FUNCTION_BLOCK pi (* 1st ordem system *)
  (* Standard: 61499-2 *)
  (* Version 11-01-12, GASR *)
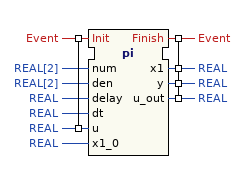
  EVENT_INPUT
    Init WITH u;
  END_EVENT
  EVENT_OUTPUT
    Finish WITH x1, y, u_out;
  END_EVENT
  VAR_INPUT
    num : ARRAY [0..1] OF REAL;
    den : ARRAY [0..1] OF REAL;
    delay : REAL := 0;
    dt : REAL;
    u : REAL;
    x1_0 : REAL; (* condicao inicial *)
  END_VAR
  VAR_OUTPUT
    x1 : REAL;
    y : REAL;
    u_out : REAL;
  END_VAR
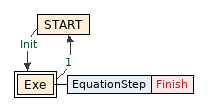
  EC_STATES
    Exe : EquationStep -> Finish;
    START;
  END_STATES
  EC_TRANSITIONS
    Exe TO START := 1;
    START TO Exe := Init;
  END_TRANSITIONS
  ALGORITHM EquationStep IN Lua: (* den[1] = b0, den[2] = b1 *)

						if type(input_buffer) ~= 'table' then
							input_buffer = {}
							for i = 1, math.ceil(delay/dt) +2 do
								input_buffer[#input_buffer +1] = 0
							end
						end
						input_buffer[#input_buffer] = u
						u = input_buffer[1]
						for i = 1, #input_buffer-1 do
							input_buffer[i] = input_buffer[i+1]
						end

						local beta1 = (num[2] - den[2]*num[1])

						local function f1(X1, U)
							return -den[2]*X1 + beta1*U
						end


						R11 = dt*f1(x1_0, u);
						x1aux = x1_0 + 0.5*R11

						R21 = dt*f1(x1aux, u);

						x1aux = x1aux + 0.5*R21

						R31 = dt*f1(x1aux, u);

						x1aux = x1aux + 0.5*R31

						R41 = dt*f1(x1aux, u);

						x1 = x1_0 + (1/6)*(R11 + 2*R21 + 2*R31 + R41)

						y  = x1 + num[1]*u

						x1_0 = x1
						if(y > 1e-12 or -y >1e-12) then
							u_out = 1/y
						end
  END_ALGORITHM
END_FUNCTION_BLOCK
(* other elements stored in the file *)
(* VarDeclaration Name=R11 Type=REAL *)
(* VarDeclaration Name=R21 Type=REAL *)
(* VarDeclaration Name=R31 Type=REAL *)
(* VarDeclaration Name=R41 Type=REAL *)
(* VarDeclaration Name=x1aux Type=REAL *)
(* VarDeclaration Name=input_buffer Type=REAL *)
